{attribute 'qualified_only'}
VAR_GLOBAL
	A : INT := 0;
END_VAR

(* stored: Version 1.1.0.1, ProductVersion 3.1.4024.16
   GVL GVL: Id {9a7287ea-6333-42eb-8a0e-d13a9195fde7} *)
